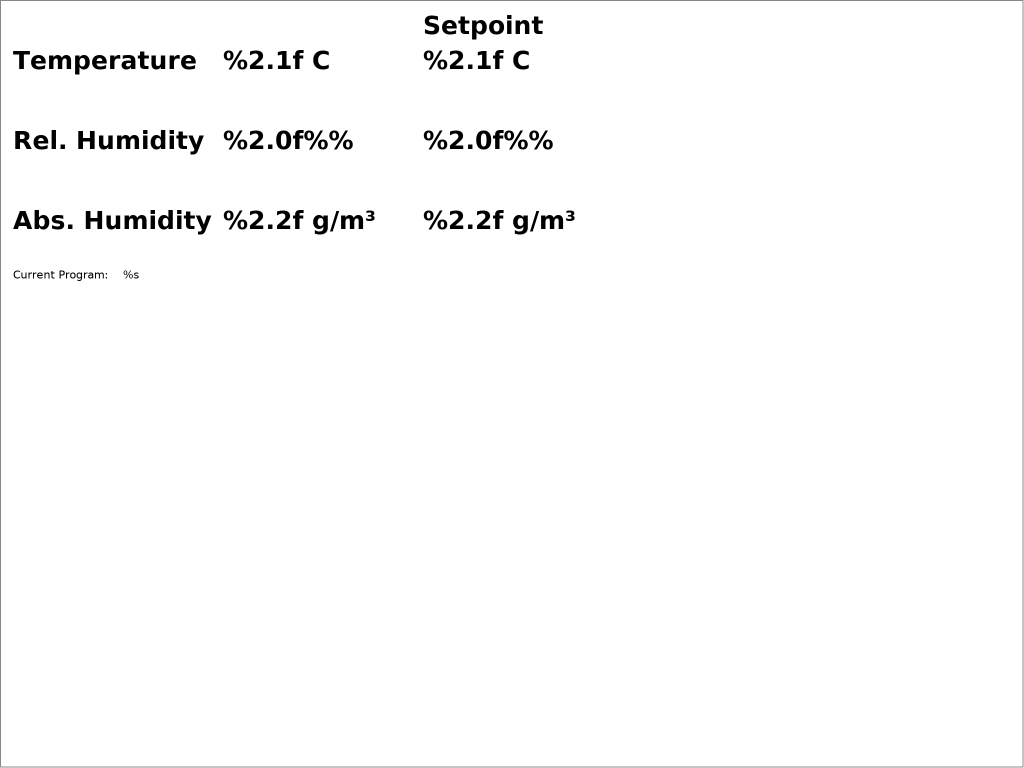
VISUALIZATION OverviewScreen  // 1024x768
    Rectangle (0,0 630x292)
    Textfield (220,40 200x40), "%2.1f C", text variable: GVL.Temp
    Textfield (420,40 200x40), "%2.1f C", text variable: GVL.TempSetpoint
    Label (10,40 200x40), "Temperature"
    Label (420,10 200x30), "Setpoint"
    Textfield (220,120 200x40), "%2.0f%%", text variable: GVL.Humidity
    Label (10,120 200x40), "Rel. Humidity"
    Textfield (120,260 120x30), "%s", text variable: GVL.CurrentProgramName
    Label (10,260 100x30), "Current Program:"
    Textfield (420,120 200x40), "%2.0f%%", text variable: GVL.HumiditySetpoint
    Textfield (220,200 200x40), "%2.2f g/m³", text variable: HumidityPID.AH
    Label (10,200 200x40), "Abs. Humidity"
    Textfield (420,200 200x40), "%2.2f g/m³", text variable: HumidityPID.AHSetpoint
END_VISUALIZATION

(* stored: Version 1.1.0.1, ProductVersion 3.1.4022.18
   Visu OverviewScreen: Id {db8952a8-2780-4596-bc64-523c746c3f36} *)
